// TIA Portal V19 export
VAR_GLOBAL   // PLC tag table "Default tag table"
   Tag_1 AT %M0.0 : Bool;
   Tag_2 AT %MW200 : Word;
   Tag_4 AT %M100.0 : Bool;
   Tag_5 AT %M100.1 : Bool;
END_VAR
